ABB RAPID module: FH24BSegmentResult.mod

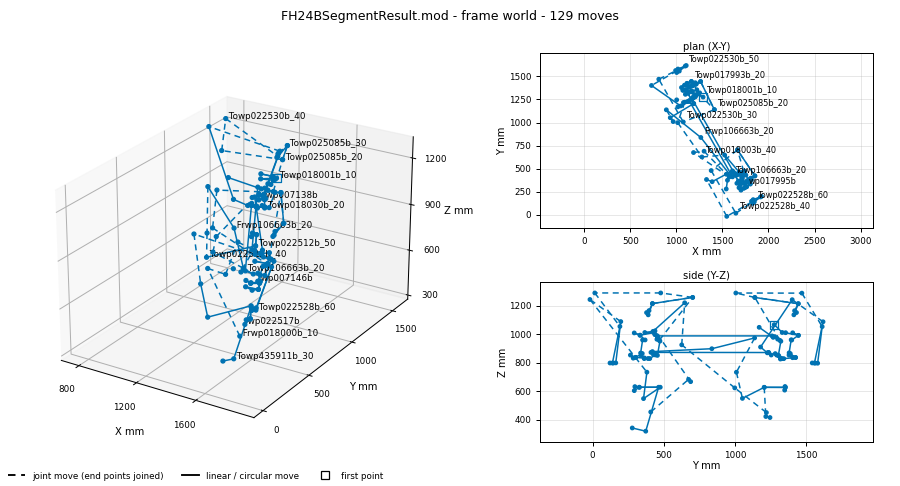
[picture p0: tool path of FH24BSegmentResult.mod in frame world, 129 of 139 moves have a stored position in this frame; points joined in program order, loops and branches not executed]
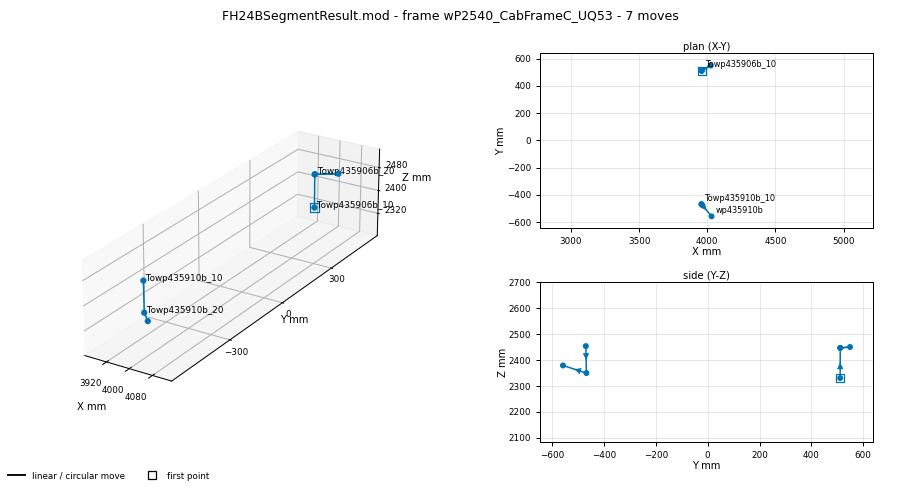
[picture p1: tool path of FH24BSegmentResult.mod in frame wP2540_CabFrameC_UQ53, 7 of 139 moves have a stored position in this frame; points joined in program order, loops and branches not executed]
%%%
  VERSION:1
  LANGUAGE:ENGLISH
%%%

MODULE FH24BSegmentA
    !# Process Simulate on eMServer 14 to ABB Rapid Volvo download
    !# ------------------------------------------------
    !# CREATED   : 27/06/2018 12:20:51 by yogesha
    !# CELL      : 2V6 Rearwall_V3
    !# ROBOT     : AR21_irb6640_235_255__d2_03
    !# PROGRAM   : FH24BSegmentA
    !# VOLP      : Abb-Rapid-Volvo 3.14.1
    !# RCS       : 5.15.02.irc5
    !# CONTROLLER: 6.0 RW6


    !# ----------------------------------------------
    !# ------ ROBTARGET
    !# ----------------------------------------------
    LOCAL CONST robtarget Towp007141b_10:=[[3996.30,641.38,1753.09],[0.331713,0.541185,0.36992,0.678403],[0,0,-3,0],[9E+09,110,9E+09,9E+09,9E+09,9E+09]];
    LOCAL CONST robtarget Towp007141b_20:=[[3995.90,593.87,1788.13],[0.283179,0.565733,0.330982,0.700137],[0,0,-3,0],[9E+09,110,9E+09,9E+09,9E+09,9E+09]];
    !
    LOCAL CONST robtarget Towp007149b_10:=[[3996.32,-641.40,1753.08],[0.331717,-0.541184,0.369916,-0.678403],[0,-1,-2,0],[9E+09,110,9E+09,9E+09,9E+09,9E+09]];
    LOCAL CONST robtarget Towp007149b_20:=[[3995.88,-593.85,1788.15],[0.283174,-0.565738,0.330987,-0.700133],[0,-1,-2,0],[9E+09,110,9E+09,9E+09,9E+09,9E+09]];
    !
    LOCAL CONST robtarget Towp017993b_10:=[[3996.22,533.94,1733.38],[0.31339,0.551104,0.355177,0.686955],[0,0,-3,0],[9E+09,110,9E+09,9E+09,9E+09,9E+09]];
    LOCAL CONST robtarget Towp017993b_20:=[[3996.30,641.37,1753.07],[0.331717,0.541178,0.36993,0.678401],[0,0,-3,0],[9E+09,110,9E+09,9E+09,9E+09,9E+09]];
    !
    LOCAL CONST robtarget Towp017994b_10:=[[3991.99,599.64,1887.87],[0.21986,0.562345,0.282351,0.745449],[0,0,-2,0],[9E+09,107.974,9E+09,9E+09,9E+09,9E+09]];
    LOCAL CONST robtarget Towp017994b_20:=[[3991.57,647.33,1916.51],[0.213228,0.580141,0.268997,0.738655],[0,0,-2,0],[9e+09,107.974,9e+09,9e+09,9e+09,9e+09]];
    LOCAL CONST robtarget Towp017994b_30:=[[4024.04,643.83,1929.61],[0.213192,0.57976,0.26894,0.738975],[0,0,-2,0],[9E+09,107.973,9E+09,9E+09,9E+09,9E+09]];
    !
    LOCAL CONST robtarget Towp017995b_10:=[[3996.22,-533.94,1733.37],[0.313389,-0.551102,0.355176,-0.686956],[0,-1,-2,0],[9E+09,110,9E+09,9E+09,9E+09,9E+09]];
    LOCAL CONST robtarget Towp017995b_20:=[[3996.32,-641.36,1753.05],[0.331718,-0.541172,0.369929,-0.678406],[0,-1,-2,0],[9E+09,110,9E+09,9E+09,9E+09,9E+09]];
    !
    LOCAL CONST robtarget Towp017996b_10:=[[3991.98,-599.64,1887.88],[0.219857,-0.562347,0.282351,-0.745448],[0,-1,-2,0],[9E+09,107.974,9E+09,9E+09,9E+09,9E+09]];
    LOCAL CONST robtarget Towp017996b_20:=[[3991.56,-647.33,1916.5],[0.213228,-0.580139,0.268997,-0.738656],[0,-1,-3,0],[9e+09,107.974,9e+09,9e+09,9e+09,9e+09]];

    LOCAL CONST robtarget Towp017996b_30:=[[4022.66,-647.20,1933.59],[0.213181,-0.579743,0.269004,-0.738969],[0,-1,-3,0],[9E+09,107.973,9E+09,9E+09,9E+09,9E+09]];
    !
    LOCAL CONST robtarget Towp435906b_10:=[[3959.73,510.86,2330.75],[0.4042,0.520538,0.419091,0.624509],[0,0,-3,0],[9E+09,116.986,9E+09,9E+09,9E+09,9E+09]];
    LOCAL CONST robtarget Towp435906b_20:=[[3959.03,511.10,2446.98],[0.315301,0.586313,0.336952,0.665787],[0,0,-3,0],[9E+09,116.986,9E+09,9E+09,9E+09,9E+09]];
    !
    LOCAL CONST robtarget Towp435905b_10:=[[3964.85,591.28,2129.79],[0.454892,0.444399,0.495034,0.592039],[0,0,-3,0],[9E+09,120.991,9E+09,9E+09,9E+09,9E+09]];
    LOCAL CONST robtarget Towp435905b_20:=[[3965.74,421.13,2129.80],[0.454868,0.444396,0.495064,0.592034],[0,0,-3,0],[9E+09,120.991,9E+09,9E+09,9E+09,9E+09]];
    LOCAL CONST robtarget Towp435905b_30:=[[3982.49,486.40,2353.36],[0.407122,0.538957,0.396041,0.622024],[0,0,-3,0],[9E+09,67.1791,9E+09,9E+09,9E+09,9E+09]];
    !
    LOCAL CONST robtarget Towp435911b_10:=[[3964.57,-591.40,2129.80],[0.523561,-0.380762,0.545621,-0.532153],[0,-1,-2,0],[9E+09,120.991,9E+09,9E+09,9E+09,9E+09]];
    LOCAL CONST robtarget Towp435911b_20:=[[3965.57,-434.58,2129.84],[0.469576,-0.431817,0.506124,-0.580392],[0,-1,-2,0],[9E+09,120.991,9E+09,9E+09,9E+09,9E+09]];
    LOCAL CONST robtarget Towp435911b_30:=[[3953.22,-482.73,2453.32],[0.299649,-0.587763,0.301228,-0.688471],[0,-1,-2,0],[9E+09,100,9E+09,9E+09,9E+09,9E+09]];
    !
    LOCAL CONST robtarget Towp435910b_10:=[[3957.78,-469.44,2453.88],[0.299678,-0.587777,0.301168,-0.688473],[0,-1,-2,0],[9E+09,150,9E+09,9E+09,9E+09,9E+09]];
    LOCAL CONST robtarget Towp435910b_20:=[[3957.17,-467.35,2350.02],[0.358354,-0.544111,0.371303,-0.661548],[0,-1,-2,0],[9E+09,106.704,9E+09,9E+09,9E+09,9E+09]];
    !
    LOCAL CONST robtarget Frwp018000b_10:=[[3966.61,-461.86,2314.83],[0.30753,-0.55023,0.279101,-0.724403],[0,-1,-2,0],[9E+09,150,9E+09,9E+09,9E+09,9E+09]];
    LOCAL CONST robtarget Frwp018000b_20:=[[4235.12,-38.76,2167.35],[0.294003,-0.458154,0.422974,-0.724387],[0,-1,-2,0],[9E+09,150,9E+09,9E+09,9E+09,9E+09]];
    !
    LOCAL CONST robtarget Towp018001b_10:=[[3997.24,431.02,1673.87],[0.244730,0.608932,0.281621,0.699992],[0,0,-2,0],[9E9,150.000,9E9,9E9,9E9,9E9]];
    !
    LOCAL CONST robtarget Towp018002b_10:=[[3991.57,647.33,1916.51],[0.213228,0.580141,0.268997,0.738655],[0,0,-2,0],[9e+09,107.974,9e+09,9e+09,9e+09,9e+09]];
    LOCAL CONST robtarget Towp018002b_20:=[[3985.46,549.99,1923.00],[0.177572,0.593147,0.183829,0.763438],[0,0,-2,0],[9E+09,107.974,9E+09,9E+09,9E+09,9E+09]];
    LOCAL CONST robtarget Towp018002b_30:=[[4032.14,551.91,1942.63],[0.171636,0.594696,0.191298,0.761754],[0,0,-2,0],[9E+09,107.974,9E+09,9E+09,9E+09,9E+09]];
    !
    LOCAL CONST robtarget Towp018003b_10:=[[3959.03,511.10,2446.98],[0.315301,0.586313,0.336952,0.665787],[0,0,-3,0],[9E+09,116.986,9E+09,9E+09,9E+09,9E+09]];
    LOCAL CONST robtarget Towp018003b_20:=[[3977.84,482.52,2322.32],[0.404341,0.520576,0.418922,0.624499],[0,0,-3,0],[9E+09,150,9E+09,9E+09,9E+09,9E+09]];
    LOCAL CONST robtarget Towp018003b_30:=[[4203.47,328.28,2218.91],[0.289162,0.516612,0.522871,0.613261],[0,0,-3,0],[9E+09,150,9E+09,9E+09,9E+09,9E+09]];
    LOCAL CONST robtarget Towp018003b_40:=[[4264.93,-125.96,1920.35],[0.0319006,-0.614182,0.118719,-0.779521],[0,-1,-3,0],[9E+09,150,9E+09,9E+09,9E+09,9E+09]];
    LOCAL CONST robtarget Towp018003b_50:=[[4152.69,-231.33,1566.84],[0.188638,-0.53985,0.266785,-0.77575],[0,-1,-3,0],[9E+09,150,9E+09,9E+09,9E+09,9E+09]];
    LOCAL CONST robtarget Towp018003b_60:=[[4035.59,-518.4,1738.81],[0.244709,-0.608865,0.281727,-0.700011],[0,-1,-3,0],[9E+09,80,9E+09,9E+09,9E+09,9E+09]];
    !
    LOCAL CONST robtarget Towp018004b_10:=[[3991.56,-647.33,1916.5],[0.213228,-0.580139,0.268997,-0.738656],[0,-1,-3,0],[9e+09,107.974,9e+09,9e+09,9e+09,9e+09]];
    LOCAL CONST robtarget Towp018004b_20:=[[3985.45,-549.99,1922.99],[0.177573,-0.593144,0.183832,-0.76344],[0,-1,-2,0],[9E+09,107.974,9E+09,9E+09,9E+09,9E+09]];
    LOCAL CONST robtarget Towp018004b_30:=[[4032.34,-551.89,1940.14],[0.171634,-0.594748,0.19138,-0.761693],[0,-1,-3,0],[9E+09,107.974,9E+09,9E+09,9E+09,9E+09]];
    !
    LOCAL CONST robtarget Towp018022b_10:=[[3966.23,-489.78,1892.65],[0.168843,-0.67567,0.149946,-0.701758],[0,-1,-3,0],[9E+09,74.9996,9E+09,9E+09,9E+09,9E+09]];
    LOCAL CONST robtarget Towp018022b_20:=[[3966.79,-489.85,1786.55],[0.235157,-0.658178,0.213799,-0.68248],[0,-1,-2,0],[9E+09,75.0003,9E+09,9E+09,9E+09,9E+09]];
    !
    LOCAL CONST robtarget Towp018024b_10:=[[4032.40,-551.87,1935.19],[0.171635,-0.594777,0.191354,-0.761677],[0,-1,-3,0],[9E+09,107.974,9E+09,9E+09,9E+09,9E+09]];
    LOCAL CONST robtarget Towp018024b_20:=[[3985.34,-535.65,1923.03],[0.177568,-0.593116,0.183807,-0.763468],[0,-1,-2,0],[9E+09,107.974,9E+09,9E+09,9E+09,9E+09]];
    LOCAL CONST robtarget Towp018024b_30:=[[3991.78,-491.36,1898.65],[0.169072,-0.675645,0.150178,-0.701677],[0,-1,-3,0],[9E+09,94.8731,9E+09,9E+09,9E+09,9E+09]];
    !
    LOCAL CONST robtarget Towp018028b_10:=[[3966.24,489.79,1892.63],[0.168846,0.675664,0.149941,0.701764],[0,0,-2,0],[9E+09,75,9E+09,9E+09,9E+09,9E+09]];
    LOCAL CONST robtarget Towp018028b_20:=[[3966.81,489.85,1786.55],[0.235157,0.658176,0.213799,0.682481],[0,0,-3,0],[9E+09,75,9E+09,9E+09,9E+09,9E+09]];
    !
    LOCAL CONST robtarget Towp018030b_10:=[[4032.39,551.86,1935.19],[0.171632,0.594777,0.191358,0.761676],[0,0,-2,0],[9E+09,107.974,9E+09,9E+09,9E+09,9E+09]];
    LOCAL CONST robtarget Towp018030b_20:=[[3985.35,535.65,1923.02],[0.177571,0.593112,0.183804,0.763471],[0,0,-2,0],[9E+09,107.974,9E+09,9E+09,9E+09,9E+09]];
    LOCAL CONST robtarget Towp018030b_30:=[[3991.79,491.35,1898.63],[0.169072,0.675639,0.150178,0.701682],[0,0,-2,0],[9E+09,94.8733,9E+09,9E+09,9E+09,9E+09]];
    !
    LOCAL CONST robtarget Towp022512b_10:=[[4073.20,471.80,1908.69],[0.242343,0.0510545,-0.0122894,-0.968761],[0,-2,-1,0],[9E+09,40.5085,9E+09,9E+09,9E+09,9E+09]];
    LOCAL CONST robtarget Towp022512b_20:=[[4356.55,510.41,1901.15],[0.303024,0.0172884,0.00682044,-0.952794],[1,-1,-1,0],[9E+09,45.3223,9E+09,9E+09,9E+09,9E+09]];
    LOCAL CONST robtarget Towp022512b_30:=[[4274.60,362.62,2127.69],[0.102237,0.586676,0.0956275,0.797621],[0,0,-2,0],[9E+09,120.001,9E+09,9E+09,9E+09,9E+09]];
    LOCAL CONST robtarget Towp022512b_40:=[[4219.28,415.22,2302.84],[0.413706,0.498371,0.323569,0.689755],[0,0,-3,0],[9E+09,120.001,9E+09,9E+09,9E+09,9E+09]];
    LOCAL CONST robtarget Towp022512b_50:=[[3965.74,421.13,2129.80],[0.454867,0.444396,0.495064,0.592035],[0,0,-3,0],[9E+09,120.991,9E+09,9E+09,9E+09,9E+09]];
    LOCAL CONST robtarget Towp022512b_60:=[[3964.85,591.28,2129.79],[0.45489,0.444399,0.495035,0.592039],[0,0,-3,0],[9E+09,120.991,9E+09,9E+09,9E+09,9E+09]];
    !
    LOCAL CONST robtarget Towp022516b_10:=[[3985.32,-804.65,1955.71],[0.0554428,0.615597,0.0620377,0.783647],[-1,0,-3,0],[9E+09,80.0001,9E+09,9E+09,9E+09,9E+09]];
    LOCAL CONST robtarget Towp022516b_20:=[[3992.76,-819.21,1650.37],[0.0414821,0.426803,0.00446797,0.903374],[-1,0,-3,0],[9E+09,120.001,9E+09,9E+09,9E+09,9E+09]];
    LOCAL CONST robtarget Towp022516b_30:=[[4454.28,-819.21,1650.39],[0.0414818,0.426789,0.00449981,0.90338],[-1,0,-3,0],[9E+09,120.001,9E+09,9E+09,9E+09,9E+09]];
    LOCAL CONST robtarget Towp022516b_40:=[[4274.61,-362.62,2127.67],[0.10224,-0.586669,0.0956253,-0.797627],[0,-1,-3,0],[9E+09,120.001,9E+09,9E+09,9E+09,9E+09]];
    LOCAL CONST robtarget Towp022516b_50:=[[4173.05,-413.61,2288.65],[0.413679,-0.498365,0.323623,-0.689751],[0,-1,-2,0],[9E+09,120.001,9E+09,9E+09,9E+09,9E+09]];
    LOCAL CONST robtarget Towp022516b_60:=[[3965.66,-421.15,2129.84],[0.464741,-0.436006,0.502516,-0.584276],[0,-1,-2,0],[9E+09,120.991,9E+09,9E+09,9E+09,9E+09]];
    LOCAL CONST robtarget Towp022516b_70:=[[3964.56,-591.39,2129.79],[0.523561,-0.380756,0.545627,-0.532152],[0,-1,-2,0],[9E+09,120.991,9E+09,9E+09,9E+09,9E+09]];
    !
    LOCAL CONST robtarget Towp022528b_10:=[[3989.55,-590.66,1514.58],[0.328179,-0.595356,0.313816,-0.662839],[0,-1,-2,0],[9E+09,120,9E+09,9E+09,9E+09,9E+09]];
    LOCAL CONST robtarget Towp022528b_20:=[[4025.67,-251.94,1481.37],[0.211082,-0.56759,0.245392,-0.757003],[0,-1,-2,0],[9E+09,120,9E+09,9E+09,9E+09,9E+09]];
    LOCAL CONST robtarget Towp022528b_30:=[[4374.56,-304.19,1572.56],[0.209509,-0.562774,0.246743,-0.760589],[0,-1,-3,0],[9E+09,120,9E+09,9E+09,9E+09,9E+09]];
    LOCAL CONST robtarget Towp022528b_40:=[[4373.35,-838.73,1572.68],[0.00204607,0.429,0.087242,0.899071],[-1,0,-3,0],[9E+09,120,9E+09,9E+09,9E+09,9E+09]];
    LOCAL CONST robtarget Towp022528b_50:=[[3992.87,-819.24,1686.63],[0.0414897,0.426835,0.00441234,0.903359],[-1,0,-3,0],[9E+09,120,9E+09,9E+09,9E+09,9E+09]];
    LOCAL CONST robtarget Towp022528b_60:=[[3985.99,-831.25,1957.00],[0.00872467,0.618253,0.0251878,0.785518],[0,-1,-3,0],[9E+09,80.0001,9E+09,9E+09,9E+09,9E+09]];
    !
    LOCAL CONST robtarget Towp022530b_10:=[[3989.52,590.65,1514.62],[0.328174,0.595365,0.313825,0.662829],[0,0,-2,0],[9E+09,120,9E+09,9E+09,9E+09,9E+09]];
    LOCAL CONST robtarget Towp022530b_20:=[[4025.65,251.95,1481.42],[0.21108,0.567605,0.245395,0.756992],[0,0,-2,0],[9E+09,120,9E+09,9E+09,9E+09,9E+09]];
    LOCAL CONST robtarget Towp022530b_30:=[[4374.56,304.20,1572.55],[0.20951,0.562772,0.246738,0.760591],[0,0,-2,0],[9E+09,120,9E+09,9E+09,9E+09,9E+09]];
    LOCAL CONST robtarget Towp022530b_40:=[[4373.38,838.72,1572.68],[0.00204401,-0.428996,0.0872399,-0.899073],[0,-1,-2,0],[9E+09,120,9E+09,9E+09,9E+09,9E+09]];
    LOCAL CONST robtarget Towp022530b_50:=[[3992.87,819.24,1686.64],[0.04149,-0.426836,0.00441444,-0.903358],[0,-1,-2,0],[9E+09,120,9E+09,9E+09,9E+09,9E+09]];
    LOCAL CONST robtarget Towp022530b_60:=[[3985.99,831.24,1957.01],[0.00872665,-0.618256,0.0251886,-0.785515],[0,0,-2,0],[9E+09,80,9E+09,9E+09,9E+09,9E+09]];
    !
    LOCAL CONST robtarget Towp025081b_10:=[[3978.83,-488.68,1784.54],[0.231134,-0.629757,0.22668,-0.706105],[0,-1,-2,0],[9E+09,130,9E+09,9E+09,9E+09,9E+09]];
    LOCAL CONST robtarget Towp025081b_20:=[[4025.67,-251.95,1481.38],[0.211082,-0.567592,0.245391,-0.757003],[0,-1,-2,0],[9E+09,120,9E+09,9E+09,9E+09,9E+09]];
    LOCAL CONST robtarget Towp025081b_30:=[[3989.53,-590.65,1514.62],[0.328174,-0.595364,0.313824,-0.662829],[0,-1,-2,0],[9E+09,120,9E+09,9E+09,9E+09,9E+09]];
    !
    LOCAL CONST robtarget Towp025085b_10:=[[3978.81,488.67,1784.54],[0.231133,0.629756,0.226682,0.706106],[0,0,-3,0],[9E+09,130,9E+09,9E+09,9E+09,9E+09]];
    LOCAL CONST robtarget Towp025085b_20:=[[4025.65,251.95,1481.41],[0.21108,0.567602,0.245394,0.756994],[0,0,-2,0],[9E+09,120,9E+09,9E+09,9E+09,9E+09]];
    LOCAL CONST robtarget Towp025085b_30:=[[3989.53,590.65,1514.61],[0.328175,0.595362,0.313824,0.662831],[0,0,-2,0],[9E+09,120,9E+09,9E+09,9E+09,9E+09]];
    LOCAL CONST robtarget Towp106661b_10:=[[3985.31,804.64,1955.73],[0.0554478,-0.615601,0.0620371,-0.783644],[0,-1,-2,0],[9E+09,80.0001,9E+09,9E+09,9E+09,9E+09]];
    LOCAL CONST robtarget Towp106661b_20:=[[3992.76,819.23,1650.39],[0.0414815,-0.426808,0.00447259,-0.903371],[0,-1,-2,0],[9E+09,120.001,9E+09,9E+09,9E+09,9E+09]];
    LOCAL CONST robtarget Towp106661b_30:=[[4454.26,819.21,1650.39],[0.0414888,-0.426792,0.00449799,-0.903378],[0,-1,-2,0],[9E+09,120.001,9E+09,9E+09,9E+09,9E+09]];
    LOCAL CONST robtarget Towp106661b_40:=[[4188.13,468.94,1908.79],[0.242334,0.0510393,-0.0123043,-0.968764],[0,-2,-1,0],[9E+09,40.8025,9E+09,9E+09,9E+09,9E+09]];
    LOCAL CONST robtarget Towp106661b_50:=[[4093.30,473.86,1918.15],[0.242338,0.0510457,-0.0122905,-0.968763],[0,-2,-1,0],[9E+09,40.8025,9E+09,9E+09,9E+09,9E+09]];
    !
    LOCAL CONST robtarget Towp106662b_10:=[[4129.59,-83.08,2146.51],[0.0379492,-0.398654,0.740598,-0.539569],[0,-1,-3,0],[9E+09,98.575,9E+09,9E+09,9E+09,9E+09]];
    LOCAL CONST robtarget Towp106662b_20:=[[4169.78,-420.74,1782.35],[0.0406723,0.23823,-0.969634,-0.0372496],[0,-1,-4,0],[9E+09,32.9298,9E+09,9E+09,9E+09,9E+09]];
    LOCAL CONST robtarget Towp106662b_30:=[[4070.84,-475.84,1774.39],[0.0406981,0.23822,-0.969635,-0.0372624],[0,-1,-4,0],[9E+09,32.9299,9E+09,9E+09,9E+09,9E+09]];
    LOCAL CONST robtarget Towp106662b_40:=[[4070.84,-475.84,1774.39],[0.0406981,0.23822,-0.969635,-0.0372624],[0,-1,-4,0],[9E+09,32.9299,9E+09,9E+09,9E+09,9E+09]];
    LOCAL CONST robtarget Frwp008446b_10:=[[4070.84,-475.84,1774.39],[0.0406981,0.23822,-0.969635,-0.0372624],[0,-1,-4,0],[9E+09,32.9299,9E+09,9E+09,9E+09,9E+09]];
    LOCAL CONST robtarget Frwp008446b_20:=[[4210.41,-357.89,1774.41],[0.04066,0.238229,-0.969635,-0.0372447],[0,-1,-4,0],[9E+09,32.9299,9E+09,9E+09,9E+09,9E+09]];
    !
    LOCAL CONST robtarget Towp106663b_10:=[[4073.20,471.79,1908.68],[0.242346,0.0510549,-0.0122924,-0.96876],[0,-2,-1,0],[9E+09,40.5084,9E+09,9E+09,9E+09,9E+09]];
    LOCAL CONST robtarget Towp106663b_20:=[[4077.25,-478.80,1910.01],[0.411397,0.0480683,-0.021155,-0.909934],[0,-2,-1,0],[9E+09,40.5089,9E+09,9E+09,9E+09,9E+09]];
    LOCAL CONST robtarget wp106663b:=[[4029.64,-483.73,1910.18],[0.381624,0.0502912,-0.019297,-0.922739],[0,-2,-1,0],[9E+09,48.5229,9E+09,9E+09,9E+09,9E+09]];
    LOCAL CONST robtarget Frwp106663b_10:=[[4089.93,-460.28,1908.57],[0.379212,0.0502876,-0.0193122,-0.923733],[0,-2,-1,0],[9E+09,40.5084,9E+09,9E+09,9E+09,9E+09]];
    LOCAL CONST robtarget Frwp106663b_20:=[[4166.11,63.29,1913.72],[0.316475,0.0499727,-0.0161716,-0.947138],[0,-2,-1,0],[9E+09,40.6758,9E+09,9E+09,9E+09,9E+09]];
    LOCAL CONST robtarget wp106664b:=[[4035.73,475.64,1776.59],[0.0438545,0.0154142,-0.998313,0.0345743],[0,-1,-4,0],[9E+09,5.69788,9E+09,9E+09,9E+09,9E+09]];
    LOCAL CONST robtarget Towp106664b_10:=[[4034.36,-472.89,1782.83],[0.0406188,0.238249,-0.969633,-0.0372129],[0,-1,-4,0],[9E+09,48.1606,9E+09,9E+09,9E+09,9E+09]];
    LOCAL CONST robtarget Towp106664b_20:=[[4082.28,-447.01,1788.74],[0.0405639,0.238266,-0.969632,-0.0371943],[0,-1,-4,0],[9E+09,96.0929,9E+09,9E+09,9E+09,9E+09]];
    LOCAL CONST robtarget Frwp106664b_10:=[[4054.41,475.57,1788.86],[0.0436763,0.0114026,-0.998369,0.034747],[0,-1,-4,0],[9E+09,109.869,9E+09,9E+09,9E+09,9E+09]];
    LOCAL CONST robtarget Frwp106664b_20:=[[4264.00,475.54,1788.87],[0.0436681,0.0114193,-0.998369,0.0347496],[0,-1,-4,0],[9E+09,109.869,9E+09,9E+09,9E+09,9E+09]];
    LOCAL CONST robtarget Towp106664b_30:=[[4077.12,478.15,1786.19],[0.043949,0.0153013,-0.998311,0.0345833],[0,-1,-4,0],[9E+09,96.0929,9E+09,9E+09,9E+09,9E+09]];
    !
    LOCAL CONST robtarget wp007138b:=[[4009.96,599.94,1888.48],[0.25778,0.662661,0.248254,0.657864],[0,0,-3,0],[9E+09,30.0008,9E+09,9E+09,9E+09,9E+09]];
    LOCAL CONST robtarget wp007141b:=[[4013.28,599.83,1792.55],[0.312947,0.639214,0.303929,0.633311],[0,0,-3,0],[9E+09,30,9E+09,9E+09,9E+09,9E+09]];
    LOCAL CONST robtarget wp017993b:=[[4071.15,637.16,1760.70],[0.381283,0.599334,0.36144,0.603961],[0,0,-3,0],[9E+09,25.0001,9E+09,9E+09,9E+09,9E+09]];
    LOCAL CONST robtarget wp017994b:=[[4068.09,637.91,1926.21],[0.241557,0.666876,0.237513,0.663701],[0,0,-2,0],[9E+09,30.0008,9E+09,9E+09,9E+09,9E+09]];
    LOCAL CONST robtarget wp435906b:=[[4025.11,548.87,2450.36],[0.337547,0.600752,0.31411,0.653055],[0,0,-3,0],[9E+09,32.614,9E+09,9E+09,9E+09,9E+09]];
    LOCAL CONST robtarget wp435905b:=[[4026.19,548.40,2376.63],[0.415469,0.554464,0.375175,0.615779],[0,0,-3,0],[9E+09,20.1716,9E+09,9E+09,9E+09,9E+09]];
    LOCAL CONST robtarget wp018001b:=[[4070.80,551.60,1758.32],[0.273553,0.647753,0.27547,0.655505],[0,0,-2,0],[9E+09,25.0008,9E+09,9E+09,9E+09,9E+09]];
    LOCAL CONST robtarget wp018002b:=[[4067.11,552.99,1929.08],[0.175428,0.674347,0.15175,0.701027],[0,0,-2,0],[9E+09,30.0023,9E+09,9E+09,9E+09,9E+09]];
    LOCAL CONST robtarget wp018028b:=[[4012.93,488.96,1787.18],[0.235151,0.658136,0.213783,0.682527],[0,0,-3,0],[9E+09,30.0003,9E+09,9E+09,9E+09,9E+09]];
    LOCAL CONST robtarget wp018030b:=[[4010.35,488.98,1894.45],[0.168846,0.675665,0.149949,0.701761],[0,0,-2,0],[9E+09,29.9998,9E+09,9E+09,9E+09,9E+09]];
    LOCAL CONST robtarget wp022512b:=[[3990.32,603.39,2132.40],[0.493157,0.490543,0.456937,0.554399],[0,0,-3,0],[9E+09,30,9E+09,9E+09,9E+09,9E+09]];
    LOCAL CONST robtarget wp022530b:=[[4015.17,829.71,1966.52],[0.0416377,-0.672562,0.0541427,-0.736873],[0,0,-2,0],[9E+09,29.9998,9E+09,9E+09,9E+09,9E+09]];
    LOCAL CONST robtarget wp022531b:=[[4015.79,805.34,1965.77],[0.0591203,-0.671069,0.0701108,-0.735691],[0,-1,-2,0],[9E+09,29.9998,9E+09,9E+09,9E+09,9E+09]];
    LOCAL CONST robtarget wp025013b:=[[3988.18,604.66,2158.61],[0.478809,0.502055,0.444253,0.56684],[0,0,-3,0],[9E+09,30.0003,9E+09,9E+09,9E+09,9E+09]];
    LOCAL CONST robtarget wp025085b:=[[4022.16,590.89,1609.19],[0.237873,0.646322,0.26848,0.673489],[0,0,-2,0],[9E+09,30.0001,9E+09,9E+09,9E+09,9E+09]];
    LOCAL CONST robtarget wp025086b:=[[4022.39,591.01,1578.79],[0.256543,0.638536,0.286361,0.666664],[0,0,-2,0],[9E+09,30.0003,9E+09,9E+09,9E+09,9E+09]];
    LOCAL CONST robtarget wp025087b:=[[4022.06,608.39,1592.15],[0.252606,0.640249,0.28259,0.668132],[0,0,-2,0],[9E+09,30.0004,9E+09,9E+09,9E+09,9E+09]];
    LOCAL CONST robtarget wp106661b:=[[4033.88,472.65,1913.14],[0.242095,0.0346761,-0.0166937,-0.969481],[0,-2,-1,0],[9E+09,40.8032,9E+09,9E+09,9E+09,9E+09]];
    LOCAL CONST robtarget wp106662b:=[[4027.51,-477.86,1777.63],[0.0405725,0.238261,-0.969633,-0.037199],[0,-1,-4,0],[9E+09,20.0007,9E+09,9E+09,9E+09,9E+09]];
    !
    LOCAL CONST robtarget wp018003b:=[[4070.50,-561.44,1759.34],[0.273524,-0.64769,0.275702,-0.655482],[0,-1,-2,0],[9E+09,24.9996,9E+09,9E+09,9E+09,9E+09]];
    LOCAL CONST robtarget wp017995b:=[[4068.32,-647.73,1761.72],[0.381249,-0.599364,0.361553,-0.603885],[0,-1,-2,0],[9E+09,25.0003,9E+09,9E+09,9E+09,9E+09]];
    LOCAL CONST robtarget wp007149b:=[[4010.31,-605.22,1793.80],[0.312926,-0.639188,0.304021,-0.633303],[0,-1,-2,0],[9E+09,30.0005,9E+09,9E+09,9E+09,9E+09]];
    LOCAL CONST robtarget wp007146b:=[[4006.40,-604.71,1889.58],[0.247896,-0.666168,0.238618,-0.661676],[0,-1,-2,0],[9E+09,30.0003,9E+09,9E+09,9E+09,9E+09]];
    LOCAL CONST robtarget wp017996b:=[[4063.78,-649.46,1925.41],[0.241507,-0.666882,0.237858,-0.66359],[0,-1,-2,0],[9E+09,29.9998,9E+09,9E+09,9E+09,9E+09]];
    LOCAL CONST robtarget wp435911b:=[[4016.24,-558.16,2451.77],[0.323471,-0.601969,0.291795,-0.669209],[0,-1,-2,0],[9E+09,19.9997,9E+09,9E+09,9E+09,9E+09]];
    LOCAL CONST robtarget wp435910b:=[[4031.57,-557.65,2379.21],[0.37943,-0.58568,0.350547,-0.624592],[0,-1,-2,0],[9E+09,29.9998,9E+09,9E+09,9E+09,9E+09]];
    LOCAL CONST robtarget wp018004b:=[[4064.49,-562.39,1927.20],[0.175404,-0.67442,0.152218,-0.700861],[0,-1,-3,0],[9E+09,30.0003,9E+09,9E+09,9E+09,9E+09]];
    LOCAL CONST robtarget wp018024b:=[[4007.58,-489.01,1894.25],[0.168841,-0.675718,0.150004,-0.701699],[0,-1,-3,0],[9E+09,30,9E+09,9E+09,9E+09,9E+09]];
    LOCAL CONST robtarget wp018022b:=[[4012.29,-489.12,1789.06],[0.235135,-0.658074,0.213939,-0.682544],[0,-1,-2,0],[9E+09,29.9996,9E+09,9E+09,9E+09,9E+09]];
    LOCAL CONST robtarget wp025081b:=[[4018.68,-590.93,1609.16],[0.218219,-0.653738,0.249811,-0.680138],[0,-1,-3,0],[9E+09,29.9996,9E+09,9E+09,9E+09,9E+09]];
    LOCAL CONST robtarget wp025080b:=[[4018.00,-590.84,1577.23],[0.256532,-0.638515,0.286499,-0.666628],[0,-1,-3,0],[9E+09,30.0003,9E+09,9E+09,9E+09,9E+09]];
    LOCAL CONST robtarget wp025082b:=[[4017.63,-608.22,1592.09],[0.252589,-0.640212,0.282689,-0.668132],[0,-1,-3,0],[9E+09,30.0008,9E+09,9E+09,9E+09,9E+09]];
    LOCAL CONST robtarget wp022528b:=[[4007.77,-837.41,1964.53],[0.0415673,0.672523,0.0539612,0.736926],[-1,-1,-3,0],[9E+09,29.9996,9E+09,9E+09,9E+09,9E+09]];
    LOCAL CONST robtarget wp022529b:=[[4008.15,-810.93,1964.86],[0.0590102,0.670958,0.0700025,0.735811],[-1,0,-3,0],[9E+09,30.0005,9E+09,9E+09,9E+09,9E+09]];
    LOCAL CONST robtarget wp022516b:=[[3987.16,-614.42,2133.13],[0.551891,-0.438963,0.522,-0.479823],[0,-1,-2,0],[9E+09,30.0005,9E+09,9E+09,9E+09,9E+09]];
    LOCAL CONST robtarget wp022517b:=[[3984.73,-615.05,2162.25],[0.541271,-0.450033,0.503418,-0.501051],[0,-1,-2,0],[9E+09,29.9998,9E+09,9E+09,9E+09,9E+09]];


    !# -----------------------------------------------
    !# ------ SPOT DATA
    !# -----------------------------------------------
    LOCAL PERS spotdata sd_wp018001b:=[15018001,0,0,0];
    LOCAL PERS spotdata sd_wp017993b:=[15017993,0,0,0];
    LOCAL PERS spotdata sd_wp007141b:=[15007141,0,0,0];
    LOCAL PERS spotdata sd_wp007138b:=[15007138,0,0,0];
    LOCAL PERS spotdata sd_wp017994b:=[15017994,0,0,0];
    LOCAL PERS spotdata sd_wp018002b:=[15018002,0,0,0];
    LOCAL PERS spotdata sd_wp018030b:=[15018030,0,0,0];
    LOCAL PERS spotdata sd_wp018028b:=[15018028,0,0,0];
    LOCAL PERS spotdata sd_wp025085b:=[15025085,0,0,0];
    LOCAL PERS spotdata sd_wp025087b:=[15025087,0,0,0];
    LOCAL PERS spotdata sd_wp025086b:=[15025086,0,0,0];
    LOCAL PERS spotdata sd_wp022530b:=[15022530,0,0,0];
    LOCAL PERS spotdata sd_wp022531b:=[15022531,0,0,0];
    LOCAL PERS spotdata sd_wp106661b:=[15106661,0,0,0];
    LOCAL PERS spotdata sd_wp106663b:=[15106663,0,0,0];
    LOCAL PERS spotdata sd_wp022512b:=[15022512,0,0,0];
    LOCAL PERS spotdata sd_wp025013b:=[15025013,0,0,0];
    LOCAL PERS spotdata sd_wp435911b:=[15435911,0,0,0];
    LOCAL PERS spotdata sd_wp018003b:=[15018003,0,0,0];
    LOCAL PERS spotdata sd_wp017995b:=[15017995,0,0,0];
    LOCAL PERS spotdata sd_wp007149b:=[15007149,0,0,0];
    LOCAL PERS spotdata sd_wp007146b:=[15007146,0,0,0];
    LOCAL PERS spotdata sd_wp017996b:=[15017996,0,0,0];
    LOCAL PERS spotdata sd_wp018004b:=[15018004,0,0,0];
    LOCAL PERS spotdata sd_wp018024b:=[15018024,0,0,0];
    LOCAL PERS spotdata sd_wp018022b:=[15018022,0,0,0];
    LOCAL PERS spotdata sd_wp025081b:=[15025081,0,0,0];
    LOCAL PERS spotdata sd_wp025082b:=[15025082,0,0,0];
    LOCAL PERS spotdata sd_wp025080b:=[15025080,0,0,0];
    LOCAL PERS spotdata sd_wp022528b:=[15022528,0,0,0];
    LOCAL PERS spotdata sd_wp022529b:=[15022529,0,0,0];
    LOCAL PERS spotdata sd_wp022516b:=[15022516,0,0,0];
    LOCAL PERS spotdata sd_wp022517b:=[15022517,0,0,0];
    LOCAL PERS spotdata sd_wp435905b:=[15435905,0,0,0];
    LOCAL PERS spotdata sd_wp106664b:=[15106664,0,0,0];
    LOCAL PERS spotdata sd_wp106662b:=[15106662,0,0,0];
    LOCAL PERS spotdata Sd_Idspot:=[246,0,0,0];
    LOCAL PERS spotdata sd_wp435906b:=[15435906,0,0,0];
    LOCAL PERS spotdata sd_wp435910b:=[15435901,0,0,0];

    !# -----------------------------------------------
    !# ------ WOBJ DATA
    !# -----------------------------------------------
    PERS wobjdata wFH24BL2_UQ51_CabFrame:=[FALSE,TRUE,"",[[5257,3059.06,1299.9],[0.164679,0.254089,-0.952025,0.0443527]],[[0,0,0],[1,0,0,0]]];




    PROC FH24B_WSeg1_A()
        MoveAbsJ HomeXQ11Gun,vmax,z100,XQ11GunTCP\WObj:=wobj0;
        MoveJ Towp018001b_10,vmax,fine,XQ11GunTCP\WObj:=wFH24BL2_UQ51_CabFrame;
        !
        SpotL wp018001b,vmax,Sd_wp018001b,XQ11Gun,XQ11GunTCP\WObj:=wFH24BL2_UQ51_CabFrame;
        !
        MoveL Towp017993b_10,vmax,z50,XQ11GunTCP\WObj:=wFH24BL2_UQ51_CabFrame;
        MoveL Towp017993b_20,vmax,fine,XQ11GunTCP\WObj:=wFH24BL2_UQ51_CabFrame;
        !
        SpotL wp017993b,vmax,Sd_wp017993b,XQ11Gun,XQ11GunTCP\WObj:=wFH24BL2_UQ51_CabFrame;
        !
        MoveL Towp007141b_10,vmax,z50,XQ11GunTCP\WObj:=wFH24BL2_UQ51_CabFrame;
        MoveL Towp007141b_20,vmax,fine,XQ11GunTCP\WObj:=wFH24BL2_UQ51_CabFrame;
        !
        SpotL wp007141b,vmax,Sd_wp007141b,XQ11Gun,XQ11GunTCP\WObj:=wFH24BL2_UQ51_CabFrame;
        SpotL wp007138b,vmax,Sd_wp007138b,XQ11Gun,XQ11GunTCP\WObj:=wFH24BL2_UQ51_CabFrame;
        !
        MoveL Towp017994b_10,vmax,z50,XQ11GunTCP\WObj:=wFH24BL2_UQ51_CabFrame;
        MoveL Towp017994b_20,vmax,z20,XQ11GunTCP\WObj:=wFH24BL2_UQ51_CabFrame;
        MoveL Towp017994b_30,vmax,fine,XQ11GunTCP\WObj:=wFH24BL2_UQ51_CabFrame;
        !
        SpotL wp017994b,vmax,Sd_wp017994b,XQ11Gun,XQ11GunTCP\WObj:=wFH24BL2_UQ51_CabFrame;
        !
        MoveL Towp018002b_10,vmax,z20,XQ11GunTCP\WObj:=wFH24BL2_UQ51_CabFrame;
        MoveL Towp018002b_20,vmax,z20,XQ11GunTCP\WObj:=wFH24BL2_UQ51_CabFrame;
        MoveL Towp018002b_30,vmax,fine,XQ11GunTCP\WObj:=wFH24BL2_UQ51_CabFrame;
        !
        SpotL wp018002b,vmax,Sd_wp018002b,XQ11Gun,XQ11GunTCP\WObj:=wFH24BL2_UQ51_CabFrame;
        !
        MoveL Towp018030b_10,vmax,z20,XQ11GunTCP\WObj:=wFH24BL2_UQ51_CabFrame;
        MoveL Towp018030b_20,vmax,z20,XQ11GunTCP\WObj:=wFH24BL2_UQ51_CabFrame;
        MoveL Towp018030b_30,vmax,fine,XQ11GunTCP\WObj:=wFH24BL2_UQ51_CabFrame;
        !
        SpotL wp018030b,vmax,Sd_wp018030b,XQ11Gun,XQ11GunTCP\WObj:=wFH24BL2_UQ51_CabFrame;
        !
        MoveL Towp018028b_10,vmax,z20,XQ11GunTCP\WObj:=wFH24BL2_UQ51_CabFrame;
        MoveL Towp018028b_20,vmax,fine,XQ11GunTCP\WObj:=wFH24BL2_UQ51_CabFrame;
        !
        SpotL wp018028b,vmax,Sd_wp018028b,XQ11Gun,XQ11GunTCP\WObj:=wFH24BL2_UQ51_CabFrame;
        !
        MoveJ Towp025085b_10,vmax,z20,XQ11GunTCP\WObj:=wFH24BL2_UQ51_CabFrame;
        MoveJ Towp025085b_20,vmax,z100,XQ11GunTCP\WObj:=wFH24BL2_UQ51_CabFrame;
        MoveL Towp025085b_30,vmax,fine,XQ11GunTCP\WObj:=wFH24BL2_UQ51_CabFrame;
        !
        SpotL wp025085b,vmax,Sd_wp025085b,XQ11Gun,XQ11GunTCP\WObj:=wFH24BL2_UQ51_CabFrame;
        SpotL wp025087b,vmax,Sd_wp025087b,XQ11Gun,XQ11GunTCP\WObj:=wFH24BL2_UQ51_CabFrame;
        SpotL wp025086b,vmax,Sd_wp025086b,XQ11Gun,XQ11GunTCP\WObj:=wFH24BL2_UQ51_CabFrame;
        !
        MoveJ Towp022530b_10,vmax,z20,XQ11GunTCP\WObj:=wFH24BL2_UQ51_CabFrame;
        MoveJ Towp022530b_20,vmax,z200,XQ11GunTCP\WObj:=wFH24BL2_UQ51_CabFrame;
        MoveJ Towp022530b_30,vmax,z200,XQ11GunTCP\WObj:=wFH24BL2_UQ51_CabFrame;
        MoveJ Towp022530b_40,vmax,z200,XQ11GunTCP\WObj:=wFH24BL2_UQ51_CabFrame;
        MoveJ Towp022530b_50,vmax,z50,XQ11GunTCP\WObj:=wFH24BL2_UQ51_CabFrame;
        MoveL Towp022530b_60,vmax,fine,XQ11GunTCP\WObj:=wFH24BL2_UQ51_CabFrame;
        !
        SpotL wp022530b,vmax,Sd_wp022530b,XQ11Gun,XQ11GunTCP\WObj:=wFH24BL2_UQ51_CabFrame;
        SpotL wp022531b,vmax,Sd_wp022531b,XQ11Gun,XQ11GunTCP\WObj:=wFH24BL2_UQ51_CabFrame;
        !
        MoveL Towp106661b_10,vmax,z50,XQ11GunTCP\WObj:=wFH24BL2_UQ51_CabFrame;
        MoveL Towp106661b_20,vmax,z50,XQ11GunTCP\WObj:=wFH24BL2_UQ51_CabFrame;
        MoveJ Towp106661b_30,vmax,z200,XQ11GunTCP\WObj:=wFH24BL2_UQ51_CabFrame;
        MoveL Towp106661b_40,vmax,z200,XQ11GunTCP\WObj:=wFH24BL2_UQ51_CabFrame;
        MoveL Towp106661b_50,vmax,fine,XQ11GunTCP\WObj:=wFH24BL2_UQ51_CabFrame;
        !
        SpotL wp106661b,v200,Sd_wp106661b\QuickRelease,XQ11Gun,XQ11GunTCP\WObj:=wFH24BL2_UQ51_CabFrame;
        !
        MoveL Towp022512b_10,vmax,z20,XQ11GunTCP\WObj:=wFH24BL2_UQ51_CabFrame;
        MoveL Towp106663b_10,vmax,z20,XQ11GunTCP\WObj:=wFH24BL2_UQ51_CabFrame;
        MoveL Towp106663b_20,vmax,fine,XQ11GunTCP\WObj:=wFH24BL2_UQ51_CabFrame;
        !
        SpotL wp106663b,v200,Sd_wp106663b\QuickRelease,XQ11Gun,XQ11GunTCP\WObj:=wFH24BL2_UQ51_CabFrame;
        !
        MoveL Frwp106663b_10,vmax,z20,XQ11GunTCP\WObj:=wFH24BL2_UQ51_CabFrame;
        MoveL Frwp106663b_20,vmax,z20,XQ11GunTCP\WObj:=wFH24BL2_UQ51_CabFrame;
        MoveL Towp022512b_20,vmax,z200,XQ11GunTCP\WObj:=wFH24BL2_UQ51_CabFrame;
        MoveJ Towp022512b_30,vmax,z200,XQ11GunTCP\WObj:=wFH24BL2_UQ51_CabFrame;
        MoveJ Towp022512b_40,vmax,z100,XQ11GunTCP\WObj:=wFH24BL2_UQ51_CabFrame;
        MoveL Towp022512b_50,vmax,z50,XQ11GunTCP\WObj:=wFH24BL2_UQ51_CabFrame;
        MoveL Towp022512b_60,vmax,fine,XQ11GunTCP\WObj:=wFH24BL2_UQ51_CabFrame;
        !
        SpotL wp022512b,vmax,Sd_wp022512b,XQ11Gun,XQ11GunTCP\WObj:=wFH24BL2_UQ51_CabFrame;
        SpotL wp025013b,vmax,Sd_wp025013b,XQ11Gun,XQ11GunTCP\WObj:=wFH24BL2_UQ51_CabFrame;
        !
        MoveL Towp435905b_10,vmax,z20,XQ11GunTCP\WObj:=wFH24BL2_UQ51_CabFrame;
        MoveL Towp435905b_20,vmax,z50,XQ11GunTCP\WObj:=wFH24BL2_UQ51_CabFrame;
        MoveJ Towp435905b_30,vmax,fine,XQ11GunTCP\WObj:=wFH24BL2_UQ51_CabFrame;
        !
        SpotL wpplate1,vmax,Sd_Idspot,XQ11Gun,XQ11GunTCP\WObj:=wobj0;
        SpotL wp435905b,vmax,Sd_wp435905b,XQ11Gun,XQ11GunTCP\WObj:=wFH24BL2_UQ51_CabFrame;
        !
        MoveL Towp435906b_10,vmax,z30,XQ11GunTCP\WObj:=wP2540_CabFrameC_UQ53;
        MoveL Towp435906b_20,vmax,fine,XQ11GunTCP\WObj:=wP2540_CabFrameC_UQ53;
        !
        SpotL wp435906b,vmax,Sd_wp435906b,XQ11Gun,XQ11GunTCP\WObj:=wP2540_CabFrameC_UQ53;
        !
        MoveL Towp018003b_10,vmax,z30,XQ11GunTCP\WObj:=wP2540_CabFrameC_UQ53;
        MoveL Towp018003b_20,vmax,z50,XQ11GunTCP\WObj:=wFH24BL2_UQ51_CabFrame;
        MoveJ Towp018003b_30,vmax,z100,XQ11GunTCP\WObj:=wFH24BL2_UQ51_CabFrame;
        MoveJ Towp018003b_40,vmax,z100,XQ11GunTCP\WObj:=wFH24BL2_UQ51_CabFrame;
        MoveJ Towp018003b_50,vmax,z100,XQ11GunTCP\WObj:=wFH24BL2_UQ51_CabFrame;
        MoveL Towp018003b_60,vmax,fine,XQ11GunTCP\WObj:=wFH24BL2_UQ51_CabFrame;
        !
        SpotL wp018003b,vmax,Sd_wp018003b,XQ11Gun,XQ11GunTCP\WObj:=wFH24BL2_UQ51_CabFrame;
        !
        MoveL Towp017995b_10,vmax,z50,XQ11GunTCP\WObj:=wFH24BL2_UQ51_CabFrame;
        MoveL Towp017995b_20,vmax,fine,XQ11GunTCP\WObj:=wFH24BL2_UQ51_CabFrame;
        !
        SpotL wp017995b,vmax,Sd_wp017995b,XQ11Gun,XQ11GunTCP\WObj:=wFH24BL2_UQ51_CabFrame;
        !
        MoveL Towp007149b_10,vmax,z50,XQ11GunTCP\WObj:=wFH24BL2_UQ51_CabFrame;
        MoveL Towp007149b_20,vmax,fine,XQ11GunTCP\WObj:=wFH24BL2_UQ51_CabFrame;
        !
        SpotL wp007149b,vmax,Sd_wp007149b,XQ11Gun,XQ11GunTCP\WObj:=wFH24BL2_UQ51_CabFrame;
        SpotL wp007146b,vmax,Sd_wp007146b,XQ11Gun,XQ11GunTCP\WObj:=wFH24BL2_UQ51_CabFrame;
        !
        MoveL Towp017996b_10,vmax,z50,XQ11GunTCP\WObj:=wFH24BL2_UQ51_CabFrame;
        MoveL Towp017996b_20,vmax,z20,XQ11GunTCP\WObj:=wFH24BL2_UQ51_CabFrame;
        MoveL Towp017996b_30,vmax,fine,XQ11GunTCP\WObj:=wFH24BL2_UQ51_CabFrame;
        !
        SpotL wp017996b,vmax,Sd_wp017996b,XQ11Gun,XQ11GunTCP\WObj:=wFH24BL2_UQ51_CabFrame;
        !
        MoveL Towp018004b_10,vmax,z20,XQ11GunTCP\WObj:=wFH24BL2_UQ51_CabFrame;
        MoveL Towp018004b_20,vmax,z20,XQ11GunTCP\WObj:=wFH24BL2_UQ51_CabFrame;
        MoveL Towp018004b_30,vmax,fine,XQ11GunTCP\WObj:=wFH24BL2_UQ51_CabFrame;
        !
        SpotL wp018004b,vmax,Sd_wp018004b,XQ11Gun,XQ11GunTCP\WObj:=wFH24BL2_UQ51_CabFrame;
        !
        MoveL Towp018024b_10,vmax,z20,XQ11GunTCP\WObj:=wFH24BL2_UQ51_CabFrame;
        MoveL Towp018024b_20,vmax,z20,XQ11GunTCP\WObj:=wFH24BL2_UQ51_CabFrame;
        MoveL Towp018024b_30,vmax,fine,XQ11GunTCP\WObj:=wFH24BL2_UQ51_CabFrame;
        !
        SpotL wp018024b,vmax,Sd_wp018024b,XQ11Gun,XQ11GunTCP\WObj:=wFH24BL2_UQ51_CabFrame;
        !
        MoveL Towp018022b_10,vmax,z20,XQ11GunTCP\WObj:=wFH24BL2_UQ51_CabFrame;
        MoveL Towp018022b_20,vmax,fine,XQ11GunTCP\WObj:=wFH24BL2_UQ51_CabFrame;
        !
        SpotL wp018022b,vmax,Sd_wp018022b,XQ11Gun,XQ11GunTCP\WObj:=wFH24BL2_UQ51_CabFrame;
        !
        MoveJ Towp025081b_10,vmax,z20,XQ11GunTCP\WObj:=wFH24BL2_UQ51_CabFrame;
        MoveJ Towp025081b_20,vmax,z100,XQ11GunTCP\WObj:=wFH24BL2_UQ51_CabFrame;
        MoveL Towp025081b_30,vmax,fine,XQ11GunTCP\WObj:=wFH24BL2_UQ51_CabFrame;
        !
        SpotL wp025081b,vmax,Sd_wp025081b,XQ11Gun,XQ11GunTCP\WObj:=wFH24BL2_UQ51_CabFrame;
        SpotL wp025082b,vmax,Sd_wp025082b,XQ11Gun,XQ11GunTCP\WObj:=wFH24BL2_UQ51_CabFrame;
        SpotL wp025080b,vmax,Sd_wp025080b,XQ11Gun,XQ11GunTCP\WObj:=wFH24BL2_UQ51_CabFrame;
        !
        MoveJ Towp022528b_10,vmax,z20,XQ11GunTCP\WObj:=wFH24BL2_UQ51_CabFrame;
        MoveJ Towp022528b_20,vmax,z200,XQ11GunTCP\WObj:=wFH24BL2_UQ51_CabFrame;
        MoveJ Towp022528b_30,vmax,z200,XQ11GunTCP\WObj:=wFH24BL2_UQ51_CabFrame;
        MoveJ Towp022528b_40,vmax,z200,XQ11GunTCP\WObj:=wFH24BL2_UQ51_CabFrame;
        MoveJ Towp022528b_50,vmax,z50,XQ11GunTCP\WObj:=wFH24BL2_UQ51_CabFrame;
        MoveL Towp022528b_60,vmax,fine,XQ11GunTCP\WObj:=wFH24BL2_UQ51_CabFrame;
        !
        SpotL wp022528b,vmax,Sd_wp022528b,XQ11Gun,XQ11GunTCP\WObj:=wFH24BL2_UQ51_CabFrame;
        SpotL wp022529b,vmax,Sd_wp022529b,XQ11Gun,XQ11GunTCP\WObj:=wFH24BL2_UQ51_CabFrame;
        !
        MoveL Towp022516b_10,vmax,z50,XQ11GunTCP\WObj:=wFH24BL2_UQ51_CabFrame;
        MoveL Towp022516b_20,vmax,z50,XQ11GunTCP\WObj:=wFH24BL2_UQ51_CabFrame;
        MoveJ Towp022516b_30,vmax,z200,XQ11GunTCP\WObj:=wFH24BL2_UQ51_CabFrame;
        MoveJ Towp022516b_40,vmax,z200,XQ11GunTCP\WObj:=wFH24BL2_UQ51_CabFrame;
        MoveL Towp022516b_50,vmax,z100,XQ11GunTCP\WObj:=wFH24BL2_UQ51_CabFrame;
        MoveL Towp022516b_60,vmax,z50,XQ11GunTCP\WObj:=wFH24BL2_UQ51_CabFrame;
        MoveL Towp022516b_70,vmax,fine,XQ11GunTCP\WObj:=wFH24BL2_UQ51_CabFrame;
        !
        SpotL wp022516b,vmax,Sd_wp022516b,XQ11Gun,XQ11GunTCP\WObj:=wFH24BL2_UQ51_CabFrame;
        SpotL wp022517b,vmax,Sd_wp022517b,XQ11Gun,XQ11GunTCP\WObj:=wFH24BL2_UQ51_CabFrame;
        !
        MoveL Towp435911b_10,vmax,z20,XQ11GunTCP\WObj:=wFH24BL2_UQ51_CabFrame;
        MoveL Towp435911b_20,vmax,z50,XQ11GunTCP\WObj:=wFH24BL2_UQ51_CabFrame;
        MoveL Towp435911b_30,vmax,fine,XQ11GunTCP\WObj:=wFH24BL2_UQ51_CabFrame;
        !
        SpotL wp435911b,vmax,Sd_wp435911b,XQ11Gun,XQ11GunTCP\WObj:=wFH24BL2_UQ51_CabFrame;
        !
        MoveL Towp435910b_10,vmax,z20,XQ11GunTCP\WObj:=wP2540_CabFrameC_UQ53;
        MoveL Towp435910b_20,vmax,fine,XQ11GunTCP\WObj:=wP2540_CabFrameC_UQ53;
        !
        SpotL wp435910b,vmax,sd_wp435910b,XQ11Gun,XQ11GunTCP\WObj:=wP2540_CabFrameC_UQ53;
        !
        MoveJ Frwp018000b_10,vmax,z50,XQ11GunTCP\WObj:=wFH24BL2_UQ51_CabFrame;
        MoveJ Frwp018000b_20,vmax,z100,XQ11GunTCP\WObj:=wFH24BL2_UQ51_CabFrame;
        MoveJ Towp106662b_10,v2000,z100,XQ11GunTCP\WObj:=wFH24BL2_UQ51_CabFrame;
        MoveJ Towp106662b_20,v2000,z100,XQ11GunTCP\WObj:=wFH24BL2_UQ51_CabFrame;
        MoveJ Towp106662b_30,v2000,z100,XQ11GunTCP\WObj:=wFH24BL2_UQ51_CabFrame;
        MoveL Towp106662b_40,v2000,fine,XQ11GunTCP\WObj:=wFH24BL2_UQ51_CabFrame;
        !
        SpotL wp106662b,v200,Sd_wp106662b\QuickRelease,XQ11Gun,XQ11GunTCP\WObj:=wFH24BL2_UQ51_CabFrame;
        !
        MoveL Towp106664b_10,vmax,z20,XQ11GunTCP\WObj:=wFH24BL2_UQ51_CabFrame;
        MoveL Towp106664b_20,vmax,z20,XQ11GunTCP\WObj:=wFH24BL2_UQ51_CabFrame;
        MoveL Towp106664b_30,vmax,fine,XQ11GunTCP\WObj:=wFH24BL2_UQ51_CabFrame;
        !
        SpotL wp106664b,v200,Sd_wp106664b\QuickRelease,XQ11Gun,XQ11GunTCP\WObj:=wFH24BL2_UQ51_CabFrame;
        !
        MoveL Frwp106664b_10,vmax,z20,XQ11GunTCP\WObj:=wFH24BL2_UQ51_CabFrame;
        MoveL Frwp106664b_20,vmax,z20,XQ11GunTCP\WObj:=wFH24BL2_UQ51_CabFrame;
        !
        MoveAbsJ HomeXQ11Gun,vmax,fine,XQ11GunTCP\WObj:=wobj0;
        RETURN ;
    ENDPROC
ENDMODULE
